{attribute 'qualified_only'}
{attribute 'strict'}
{attribute 'to_string'}
TYPE E_HE_SolidAttenuatorSlotState :
(
    FULL := 0,
    EMPTY
) INT;
END_TYPE

(* stored: Version 1.1.0.1
   DUT E_HE_SolidAttenuatorSlotState: Id {661fb182-1eac-4a51-90bc-b162621932bd} *)
